Staubli VAL3: insertValue.pgx

program insertValue(num& x_nValue[] (dimensions=1), num x_nIndex (dimensions=1))
begin
  if nDistance[0]!=-1
    // insert
    insert(nDistance[x_nIndex])
    insert(nCoeff[x_nIndex])
    insert(nJoint[x_nIndex])
    insert(nHome[x_nIndex])
  endIf
  // copy
  nCoeff[x_nIndex]=x_nValue[3]
  nDistance[x_nIndex]=x_nValue[2]
  nJoint[x_nIndex]=x_nValue[1]
  nHome[x_nIndex]=x_nValue
end
